FUNCTION_BLOCK FB_SendTargetVelocity_Left
VAR_INPUT
	TargetVelocity : LREAL;
END_VAR
VAR_OUTPUT
END_VAR
VAR
	TxMessage : EXTCANQUEUE;
	i : INT;
	TargetVelocity_Values : ARRAY[0..1] OF BYTE;
END_VAR
VAR_IN_OUT
	CAN_OUTPUTS_Left : CANTXQUEUESTRUCT_E_32;
	CAN_INPUTS_Left : CANRXQUEUESTRUCT_E_32;
END_VAR

TargetVelocity_Values[1] := INT_TO_BYTE(LREAL_TO_INT(TargetVelocity) AND 16#FF);
TargetVelocity_Values[0] := INT_TO_BYTE(SHR(LREAL_TO_INT(TargetVelocity), 8) AND 16#FF);


TxMessage.cobId := 300;
TxMessage.length := 2;
FOR i := 0 TO 1 DO 
		TxMessage.data[i] := TargetVelocity_Values[i];
END_FOR
CAN_OUTPUTS_Left.TxMessages[8] := TxMessage;
//CAN_OUTPUTS.NoOfTxMessages := 1;

END_FUNCTION_BLOCK

(* stored: Version 1.1.0.1
   POU FB_SendTargetVelocity_Left: Id {64d14829-60c2-4275-ba28-2e7fd7a4ef7c}, SpecialFunc None *)
